FUNCTION Convert_LWORD_TO_DT : BOOL
VAR_INPUT
	in : LWORD;
	out : REFERENCE TO DT;
END_VAR
VAR
	converted : DT;
END_VAR

converted := LWORD_TO_DT(in);

IF (DT_TO_LWORD(converted) <> in) THEN
	RETURN;
END_IF

out := converted;
Convert_LWORD_TO_DT := TRUE;

END_FUNCTION

(* stored: Version 1.1.0.1, ProductVersion 3.1.4024.12
   POU Convert_LWORD_TO_DT: Id {7344f749-9f9b-4026-8d90-8d405e653283}, SpecialFunc None *)
